FUNCTION_BLOCK FB_Running
VAR_INPUT
	bManual : BOOL;
	bStart : BOOL;
	bStop : BOOL;
	bAuto : BOOL;
END_VAR
VAR_OUTPUT
	bRunning : BOOL;
	bAutoMode : BOOL;
	bManualMode : BOOL;
END_VAR
VAR
END_VAR


IF NOT(bStart) AND NOT(bManual) AND NOT(bAuto) OR (bStop) THEN
	bRunning := FALSE;
	bAutoMode := FALSE;
	bManualMode := FALSE;	
	
ELSIF bStart AND bAuto AND NOT(bStop) THEN
	bRunning := TRUE;
	bAutoMode := TRUE;
	bManualMode := FALSE;
	
ELSIF bStart AND bManual AND NOT(bStop) THEN
	bRunning := TRUE;
	bManualMode := TRUE;
	bAutoMode := FALSE;
END_IF

END_FUNCTION_BLOCK

(* stored: Version 1.1.0.1
   POU FB_Running: Id {0482d1f2-7e27-4274-b9ba-9a1a0424916f}, SpecialFunc None *)
